FUNCTION_BLOCK NotBindTest EXTENDS TcUnit.FB_TestSuite

BindAndTestBinding();

METHOD BindAndTestBinding : BOOL
VAR
	expected : BOOL;
	actual : BOOL;
	
	variable : BOOL;
	binding : BoolValue;
	disposable : Disposable;
END_VAR
TcUnit.TEST('Bind and test binding');

binding := NotBind(variable);

expected := TRUE;
actual := binding <> 0;

AssertEquals(
	Expected := expected,
	Actual := actual,
	Message := 'NotBind should return interface to created Binding');
	
variable := FALSE;

expected := TRUE;
actual := binding.Value;

AssertEquals(
	Expected := expected,
	Actual := actual,
	Message := 'Binding should return negated value of binded variable');
	
__QUERYINTERFACE(binding, disposable);
disposable.Dispose();

TEST_FINISHED();
END_METHOD

END_FUNCTION_BLOCK

(* stored: Version 1.1.0.1, ProductVersion 3.1.4024.12
   POU NotBindTest: Id {fe96cbef-b99a-0478-3f0f-27ee3f2d8f78}, SpecialFunc None
   Method BindAndTestBinding: Id {98850e43-29ab-0cbc-258e-5c83ac52f810} *)
